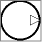
VISUALIZATION VISU_M1Figure_Supply  // 42x42
    Ellipse (0,0 40x40)
    Polygon (30,25) (40,20) (30,15)
END_VISUALIZATION

(* stored: Version 1.1.0.1, ProductVersion 3.1.4018.2
   Visu VISU_M1Figure_Supply: Id {3f4cbc65-ba76-4152-95bb-21c230d9f13e} *)
